INTERFACE ITF_BaseLocation

END_INTERFACE

(* stored: Version 1.1.0.1
   Itf ITF_BaseLocation: Id {ccad8ee0-a020-06c4-1cac-6daab23bc46c} *)
